RESOURCE_TYPE _CBCore0
  (* Standard: 61499-2 *)
  (* Version 0.1, 2019-00-29, hpea485, UOA *)
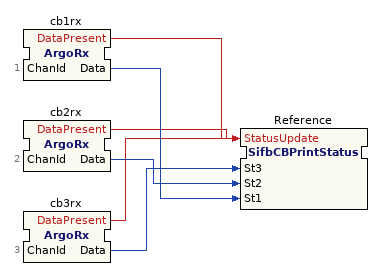
  FBS
    cb3rx : ArgoRx(ChanId := 3);
    cb2rx : ArgoRx(ChanId := 2);
    cb1rx : ArgoRx(ChanId := 1);
    Reference : SifbCBPrintStatus;
  END_FBS
  EVENT_CONNECTIONS
    cb3rx.DataPresent TO Reference.StatusUpdate;
    cb2rx.DataPresent TO Reference.StatusUpdate;
    cb1rx.DataPresent TO Reference.StatusUpdate;
  END_CONNECTIONS
  DATA_CONNECTIONS
    cb3rx.Data TO Reference.St3;
    cb2rx.Data TO Reference.St2;
    cb1rx.Data TO Reference.St1;
  END_CONNECTIONS
END_RESOURCE_TYPE
